// TIA Portal project "sova on" (V17)

(* hardware
DEVICE "S7-1200 station_1"  S7-1200 Station
   slot 0: "Rack_0"  S7-1200 Rack  Rack  V1.0
   slot 1: "D1_PLC"  CPU 1214C DC/DC/DC  6ES7 214-1AG40-0XB0  V4.4
   slot 2: "D2_16x24VDC/DQ16xRelay"  SM 1223 DI16/DQ16 x relay  6ES7 223-1PL32-0XB0  V2.0
   slot 3: "DI 8/DQ 8x24VDC_1"  6ES7 223-1BH32-0XB0  V2.0
   slot 4: "AI 8x13BIT_1"  6ES7 231-4HF32-0XB0  V2.1
   slot 5: "AI 4x13BIT_1"  6ES7 231-4HD32-0XB0  V2.1
   slot 101: "D0.1_CM 1241"  6ES7 241-1CH32-0XB0  V2.2
   slot 102: "D0.2_CM 1241"  6ES7 241-1CH32-0XB0  V2.2
*)

// ===== PLC "D1_PLC"  CPU 1214C DC/DC/DC =====

VAR_GLOBAL   // PLC tag table "Default tag table"
   "System_Byte" AT %MB1 : Byte;
   "FirstScan" AT %M1.0 : Bool;
   "DiagStatusUpdate" AT %M1.1 : Bool;
   "AlwaysTRUE" AT %M1.2 : Bool;
   "AlwaysFALSE" AT %M1.3 : Bool;
   "Clock_Byte" AT %MB0 : Byte;
   "Clock_10Hz" AT %M0.0 : Bool;
   "Clock_5Hz" AT %M0.1 : Bool;
   "Clock_2.5Hz" AT %M0.2 : Bool;
   "Clock_2Hz" AT %M0.3 : Bool;
   "Clock_1.25Hz" AT %M0.4 : Bool;
   "Clock_1Hz" AT %M0.5 : Bool;
   "Clock_0.625Hz" AT %M0.6 : Bool;
   "Clock_0.5Hz" AT %M0.7 : Bool;
END_VAR

VAR_GLOBAL   // PLC tag table "SOVA"
   "Write_tags" AT %MW4002 : Word;
END_VAR

VAR_GLOBAL   // PLC tag table "DQ"
   "DQa1.0" AT %Q0.0 : Bool;
   "DQa1.1" AT %Q0.1 : Bool;
   "DQa1.2" AT %Q0.2 : Bool;
   "DQa1.3" AT %Q0.3 : Bool;
   "DQa1.4" AT %Q0.4 : Bool;
   "DQa1.5" AT %Q0.5 : Bool;
   "DQa1.6" AT %Q0.6 : Bool;
   "DQa1.7" AT %Q0.7 : Bool;
   "DQb1.0" AT %Q1.0 : Bool;
   "DQb1.1" AT %Q1.1 : Bool;
   "RQa2.0" AT %Q8.0 : Bool;
   "RQa2.1" AT %Q8.1 : Bool;
   "RQa2.2" AT %Q8.2 : Bool;
   "RQa2.3" AT %Q8.3 : Bool;
   "RQa2.4" AT %Q8.4 : Bool;
   "RQa2.5" AT %Q8.5 : Bool;
   "RQa2.6" AT %Q8.6 : Bool;
   "RQa2.7" AT %Q8.7 : Bool;
   "RQb2.0" AT %Q9.0 : Bool;
   "RQb2.1" AT %Q9.1 : Bool;
   "RQb2.2" AT %Q9.2 : Bool;
   "RQb2.3" AT %Q9.3 : Bool;
   "RQb2.4" AT %Q9.4 : Bool;
   "RQb2.5" AT %Q9.5 : Bool;
   "RQb2.6" AT %Q9.6 : Bool;
   "RQb2.7" AT %Q9.7 : Bool;
   "DQa3.0" AT %Q12.0 : Bool;
   "DQa3.1" AT %Q12.1 : Bool;
   "DQa3.2" AT %Q12.2 : Bool;
   "DQa3.3" AT %Q12.3 : Bool;
   "DQa3.4" AT %Q12.4 : Bool;
   "DQa3.5" AT %Q12.5 : Bool;
   "DQa3.6" AT %Q12.6 : Bool;
   "DQa3.7" AT %Q12.7 : Bool;
   "DQb3.0" AT %Q13.0 : Bool;
   "DQb3.1" AT %Q13.1 : Bool;
   "DQb3.2" AT %Q13.2 : Bool;
   "DQb3.3" AT %Q13.3 : Bool;
   "DQb3.4" AT %Q13.4 : Bool;
   "DQb3.5" AT %Q13.5 : Bool;
   "DQb3.6" AT %Q13.6 : Bool;
   "DQb3.7" AT %Q13.7 : Bool;
   "DQa4.0" AT %Q16.0 : Bool;
   "DQa4.1" AT %Q16.1 : Bool;
   "DQa4.2" AT %Q16.2 : Bool;
   "DQa4.3" AT %Q16.3 : Bool;
   "DQa4.4" AT %Q16.4 : Bool;
   "DQa4.5" AT %Q16.5 : Bool;
   "DQa4.6" AT %Q16.6 : Bool;
   "DQa4.7" AT %Q16.7 : Bool;
   "DQb4.0" AT %Q17.0 : Bool;
   "DQb4.1" AT %Q17.1 : Bool;
   "DQb4.2" AT %Q17.2 : Bool;
   "DQb4.3" AT %Q17.3 : Bool;
   "DQb4.4" AT %Q17.4 : Bool;
   "DQb4.5" AT %Q17.5 : Bool;
   "DQb4.6" AT %Q17.6 : Bool;
   "DQb4.7" AT %Q17.7 : Bool;
   "DQa5.0" AT %Q20.0 : Bool;
   "DQa5.1" AT %Q20.1 : Bool;
   "DQa5.2" AT %Q20.2 : Bool;
   "DQa5.3" AT %Q20.3 : Bool;
   "DQa5.4" AT %Q20.4 : Bool;
   "DQa5.5" AT %Q20.5 : Bool;
   "DQa5.6" AT %Q20.6 : Bool;
   "DQa5.7" AT %Q20.7 : Bool;
   "DQb5.0" AT %Q21.0 : Bool;
   "DQb5.1" AT %Q21.1 : Bool;
   "DQb5.2" AT %Q21.2 : Bool;
   "DQb5.3" AT %Q21.3 : Bool;
   "DQb5.4" AT %Q21.4 : Bool;
   "DQb5.5" AT %Q21.5 : Bool;
   "DQb5.6" AT %Q21.6 : Bool;
   "DQb5.7" AT %Q21.7 : Bool;
END_VAR

VAR_GLOBAL   // PLC tag table "AI"
   "AI7.0" AT %IW144 : Int;
   "AI7.1" AT %IW146 : Int;
   "AI7.2" AT %IW148 : Int;
   "AI7.3" AT %IW150 : Int;
   "AI7.4" AT %IW152 : Int;
   "AI7.5" AT %IW154 : Int;
   "AI7.6" AT %IW156 : Int;
   "AI7.7" AT %IW158 : Int;
   "AI8.0" AT %IW160 : Int;
   "AI8.1" AT %IW162 : Int;
   "AI8.2" AT %IW164 : Int;
   "AI8.3" AT %IW166 : Int;
   "AI8.4" AT %IW168 : Int;
   "AI8.5" AT %IW170 : Int;
   "AI8.6" AT %IW172 : Int;
   "AI8.7" AT %IW174 : Int;
END_VAR

DATA_BLOCK "Data_block_1"   // DB1
{ S7_Optimized_Access := 'TRUE' }
VERSION : 0.1
   VAR
      "DQa1.0" : Bool;
      "DQa1.1" : Bool;
      "DQa1.2" : Bool;
      "DQa1.3" : Bool;
      "DQa1.4" : Bool;
      "DQa1.5" : Bool;
      "DQa1.6" : Bool;
      "DQa1.7" : Bool;
      "DQb1.0" : Bool;
      "DQb1.1" : Bool;
      "RQa2.0" : Bool;
      "RQa2.1" : Bool;
      "RQa2.2" : Bool;
      "RQa2.3" : Bool;
      "RQa2.4" : Bool;
      "RQa2.5" : Bool;
      "RQa2.6" : Bool;
      "RQa2.7" : Bool;
      "RQb2.0" : Bool;
      "RQb2.1" : Bool;
      "RQb2.2" : Bool;
      "RQb2.3" : Bool;
      "RQb2.4" : Bool;
      "RQb2.5" : Bool;
      "RQb2.6" : Bool;
      "RQb2.7" : Bool;
      "DQa3.0" : Bool;
      "DQa3.1" : Bool;
      "DQa3.2" : Bool;
      "DQa3.3" : Bool;
      "DQa3.4" : Bool;
      "DQa3.5" : Bool;
      "DQa3.6" : Bool;
      "DQa3.7" : Bool;
      "DQb3.0" : Bool;
      "DQb3.1" : Bool;
      "DQb3.2" : Bool;
      "DQb3.3" : Bool;
      "DQb3.4" : Bool;
      "DQb3.5" : Bool;
      "DQb3.6" : Bool;
      "DQb3.7" : Bool;
      "DQa4.0" : Bool;
      "DQa4.1" : Bool;
      "DQa4.2" : Bool;
      "DQa4.3" : Bool;
      "DQa4.4" : Bool;
      "DQa4.5" : Bool;
      "DQa4.6" : Bool;
      "DQa4.7" : Bool;
      "DQb4.0" : Bool;
      "DQb4.1" : Bool;
      "DQb4.2" : Bool;
      "DQb4.3" : Bool;
      "DQb4.4" : Bool;
      "DQb4.5" : Bool;
      "DQb4.6" : Bool;
      "DQb4.7" : Bool;
      "DQa5.0" : Bool;
      "DQa5.1" : Bool;
      "DQa5.2" : Bool;
      "DQa5.3" : Bool;
      "DQa5.4" : Bool;
      "DQa5.5" : Bool;
      "DQa5.6" : Bool;
      "DQa5.7" : Bool;
      "DQb5.0" : Bool;
      "DQb5.1" : Bool;
      "DQb5.2" : Bool;
      "DQb5.3" : Bool;
      "DQb5.4" : Bool;
      "DQb5.5" : Bool;
      "DQb5.6" : Bool;
      "DQb5.7" : Bool;
      "DQa6.0" : Bool;
      "DQa6.1" : Bool;
      "DQa6.2" : Bool;
      "DQa6.3" : Bool;
      "DQa6.4" : Bool;
      "DQa6.5" : Bool;
      "DQa6.6" : Bool;
      "DQa6.7" : Bool;
      "DQb6.0" : Bool;
      "DQb6.1" : Bool;
      "DQb6.2" : Bool;
      "DQb6.3" : Bool;
      "DQb6.4" : Bool;
      "DQb6.5" : Bool;
      "DQb6.6" : Bool;
      "DQb6.7" : Bool;
   END_VAR
BEGIN
END_DATA_BLOCK

DATA_BLOCK "SOVA_first_run_DB_1"   // DB2
{ S7_Optimized_Access := 'TRUE' }
VERSION : 0.1
// stored: InstanceOfName SOVA_first_run
"SOVA_first_run"
BEGIN
END_DATA_BLOCK

DATA_BLOCK "SOVA_onoff_DB_1"   // DB3
{ S7_Optimized_Access := 'TRUE' }
VERSION : 0.1
// stored: InstanceOfName SOVA_onoff
"SOVA_onoff"
BEGIN
END_DATA_BLOCK

DATA_BLOCK "SOVA_first_run_DB_2"   // DB4
{ S7_Optimized_Access := 'TRUE' }
VERSION : 0.1
// stored: InstanceOfName SOVA_first_run
"SOVA_first_run"
BEGIN
END_DATA_BLOCK

DATA_BLOCK "ModbusMasterConnector_DB_1"   // DB94
{ S7_Optimized_Access := 'FALSE' }
VERSION : 0.1
// stored: InstanceOfName ModbusMasterConnector
"ModbusMasterConnector"
BEGIN
END_DATA_BLOCK

DATA_BLOCK "SOVA_first_run_DB"   // DB98
{ S7_Optimized_Access := 'TRUE' }
VERSION : 0.1
// stored: InstanceOfName SOVA_first_run
"SOVA_first_run"
BEGIN
END_DATA_BLOCK

DATA_BLOCK "SOVA_onoff_DB"   // DB179
{ S7_Optimized_Access := 'TRUE' }
VERSION : 0.1
// stored: InstanceOfName SOVA_onoff
"SOVA_onoff"
BEGIN
END_DATA_BLOCK

FUNCTION_BLOCK "ModbusMasterConnector"   // FB12, SCL
{ S7_Optimized_Access := 'FALSE' }
VERSION : 0.1
   VAR_INPUT
      Total_devices : Int;
      port_1 : Hw_SubModule;
   END_VAR
   VAR
      instModbusCommLoad : Modbus_Comm_Load;
      instModbusMaster : Modbus_Master;
      init : Bool := True;
      PORT : Port := 269;
      BAUD : UDInt := 9600;
      STOP_BITS : USInt := 1;
      PARITY : UInt;
      Read_REGS : Word;
      "Step" : UInt;
      Write_REGS : Array[0..10] of Word;
   END_VAR
   VAR_TEMP
      "Counter" : Int;
   END_VAR
BEGIN
   IF #init THEN
       #Step := 2;
       #instModbusCommLoad.MODE := 4;
       #instModbusCommLoad.STOP_BITS := #STOP_BITS;
   END_IF;

   #instModbusCommLoad(REQ := #init,
                       "PORT" := #port_1,
                       BAUD := #BAUD,
                       PARITY := #PARITY,
                       MB_DB := #instModbusMaster.MB_DB);

   #init := FALSE;

           FOR #Counter := 1 TO #Total_devices DO
               #instModbusMaster(REQ := TRUE,
                                 MB_ADDR := #Counter,
                                 MODE := 1,
                                 DATA_ADDR := 40002,
                                 DATA_LEN := 1,
                                 DATA_PTR := "Write_tags");
               ;
           END_FOR;
END_FUNCTION_BLOCK

FUNCTION_BLOCK "SOVA_onoff"   // FB16, SCL
{ S7_Optimized_Access := 'TRUE' }
VERSION : 0.1
   VAR_INPUT
      Device_total : Int;
      Port : Hw_SubModule;
   END_VAR
   VAR
      www : Word := 16#F7C0;
   END_VAR
   VAR_TEMP
      "Counter" : Int;
      Master_reading_done : Bool;
      Sova_input_counter : Int;
      COMM_LOAD_DONE : Bool;
   END_VAR
BEGIN
   "MB_COMM_LOAD_DB"(REQ:="FirstScan",
                     "PORT":=#Port,
                     BAUD:=9600,
                     DONE=>#COMM_LOAD_DONE,
                     MB_DB:="MB_MASTER_DB");


   IF #COMM_LOAD_DONE THEN
       "MB_MASTER_DB"(REQ := TRUE,
                      MB_ADDR := 2,
                      MODE := 1,
                      DATA_ADDR := 40002,
                      DONE => #Master_reading_done,
                      DATA_LEN := 1,
                      DATA_PTR := #www);
   END_IF;
END_FUNCTION_BLOCK

FUNCTION_BLOCK "SOVA_first_run"   // FB17, SCL
{ S7_Optimized_Access := 'TRUE' }
VERSION : 0.1
BEGIN
   "Write_tags".%X0 := 1;
   "Write_tags".%X1 := 1;
   "Write_tags".%X2 := 1;
   "Write_tags".%X3 := 1;
   "Write_tags".%X4 := 1;
   "Write_tags".%X5 := 1;
   "Write_tags".%X6 := 1;
   "Write_tags".%X7 := 1;
   "Write_tags".%X8 := 1;
   "Write_tags".%X9 := 1;
   "Write_tags".%X10:= 1;
   "Write_tags".%X11:= 1;
END_FUNCTION_BLOCK

ORGANIZATION_BLOCK "Main"   // OB1, LAD, ProgramCycle
TITLE = "Main Program Sweep (Cycle)"
{ S7_Optimized_Access := 'TRUE' }
VERSION : 0.1
   VAR_INPUT
      Initial_Call : Bool;   // Initial call of this OB
      Remanence : Bool;   // =True, if remanent data are available
   END_VAR
   VAR_TEMP   // added for the SCL form of the ladder/FBD networks
      _w1 : Bool;
   END_VAR
BEGIN

REGION Network 1: MODBUS
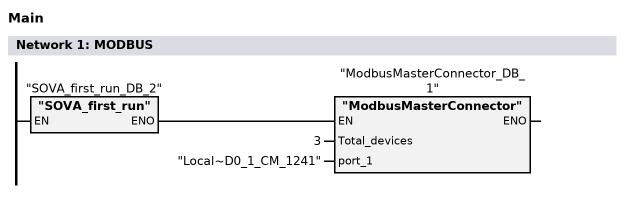
   RUNG wire#powerrail
      "SOVA_first_run_DB_2"()
      "ModbusMasterConnector_DB_1"(Total_devices := 3, port_1 := "Local~D0_1_CM_1241")
   END_RUNG
   // the same network as SCL:
   "SOVA_first_run_DB_2"(ENO => #_w1);   // "SOVA_first_run"
   IF #_w1 THEN
       "ModbusMasterConnector_DB_1"(Total_devices := 3, port_1 := "Local~D0_1_CM_1241");   // "ModbusMasterConnector"
   END_IF;
END_REGION

REGION Network 3 (SCL)
   "DQa1.0" := "Data_block_1"."DQa1.0";
   "DQa1.1" := "Data_block_1"."DQa1.1";
   "DQa1.2" := "Data_block_1"."DQa1.2";
   "DQa1.3" := "Data_block_1"."DQa1.3";
   "DQa1.4" := "Data_block_1"."DQa1.4";
   "DQa1.5" := "Data_block_1"."DQa1.5";
   "DQa1.6" := "Data_block_1"."DQa1.6";
   "DQa1.7" := "Data_block_1"."DQa1.7";
   "DQb1.0" := "Data_block_1"."DQb1.0";
   "DQb1.1" := "Data_block_1"."DQb1.1";
   "RQa2.0" := "Data_block_1"."RQa2.0";
   "RQa2.1" := "Data_block_1"."RQa2.1";
   "RQa2.2" := "Data_block_1"."RQa2.2";
   "RQa2.3" := "Data_block_1"."RQa2.3";
   "RQa2.4" := "Data_block_1"."RQa2.4";
   "RQa2.5" := "Data_block_1"."RQa2.5";
   "RQa2.6" := "Data_block_1"."RQa2.6";
   "RQa2.7" := "Data_block_1"."RQa2.7";
   "RQb2.0" := "Data_block_1"."RQb2.0";
   "RQb2.1" := "Data_block_1"."RQb2.1";
   "RQb2.2" := "Data_block_1"."RQb2.2";
   "RQb2.3" := "Data_block_1"."RQb2.3";
   "RQb2.4" := "Data_block_1"."RQb2.4";
   "RQb2.5" := "Data_block_1"."RQb2.5";
   "RQb2.6" := "Data_block_1"."RQb2.6";
   "RQb2.7" := "Data_block_1"."RQb2.7";
   "DQa3.0" := "Data_block_1"."DQa3.0";
   "DQa3.1" := "Data_block_1"."DQa3.1";
   "DQa3.2" := "Data_block_1"."DQa3.2";
   "DQa3.3" := "Data_block_1"."DQa3.3";
   "DQa3.4" := "Data_block_1"."DQa3.4";
   "DQa3.5" := "Data_block_1"."DQa3.5";
   "DQa3.6" := "Data_block_1"."DQa3.6";
   "DQa3.7" := "Data_block_1"."DQa3.7";
   "DQb3.0" := "Data_block_1"."DQb3.0";
   "DQb3.1" := "Data_block_1"."DQb3.1";
   "DQb3.2" := "Data_block_1"."DQb3.2";
   "DQb3.3" := "Data_block_1"."DQb3.3";
   "DQb3.4" := "Data_block_1"."DQb3.4";
   "DQb3.5" := "Data_block_1"."DQb3.5";
   "DQb3.6" := "Data_block_1"."DQb3.6";
   "DQb3.7" := "Data_block_1"."DQb3.7";
   "DQa4.0" := "Data_block_1"."DQa4.0";
   "DQa4.1" := "Data_block_1"."DQa4.1";
   "DQa4.2" := "Data_block_1"."DQa4.2";
   "DQa4.3" := "Data_block_1"."DQa4.3";
   "DQa4.4" := "Data_block_1"."DQa4.4";
   "DQa4.5" := "Data_block_1"."DQa4.5";
   "DQa4.6" := "Data_block_1"."DQa4.6";
   "DQa4.7" := "Data_block_1"."DQa4.7";
   "DQb4.0" := "Data_block_1"."DQb4.0";
   "DQb4.1" := "Data_block_1"."DQb4.1";
   "DQb4.2" := "Data_block_1"."DQb4.2";
   "DQb4.3" := "Data_block_1"."DQb4.3";
   "DQb4.4" := "Data_block_1"."DQb4.4";
   "DQb4.5" := "Data_block_1"."DQb4.5";
   "DQb4.6" := "Data_block_1"."DQb4.6";
   "DQb4.7" := "Data_block_1"."DQb4.7";
   "DQa5.0" := "Data_block_1"."DQa5.0";
   "DQa5.1" := "Data_block_1"."DQa5.1";
   "DQa5.2" := "Data_block_1"."DQa5.2";
   "DQa5.3" := "Data_block_1"."DQa5.3";
   "DQa5.4" := "Data_block_1"."DQa5.4";
   "DQa5.5" := "Data_block_1"."DQa5.5";
   "DQa5.6" := "Data_block_1"."DQa5.6";
   "DQa5.7" := "Data_block_1"."DQa5.7";
   "DQb5.0" := "Data_block_1"."DQb5.0";
   "DQb5.1" := "Data_block_1"."DQb5.1";
   "DQb5.2" := "Data_block_1"."DQb5.2";
   "DQb5.3" := "Data_block_1"."DQb5.3";
   "DQb5.4" := "Data_block_1"."DQb5.4";
   "DQb5.5" := "Data_block_1"."DQb5.5";
   "DQb5.6" := "Data_block_1"."DQb5.6";
   "DQb5.7" := "Data_block_1"."DQb5.7";
END_REGION
END_ORGANIZATION_BLOCK